// SIMATIC S7-200 project (STEP 7-Micro/WIN), CPU 224 REL 01.11

SYMBOL_TABLE USER1
Onn              I0.0
Off              I0.1
END_SYMBOL_TABLE

ORGANIZATION_BLOCK MAIN:OB1
TITLE=PROGRAM COMMENTS
BEGIN
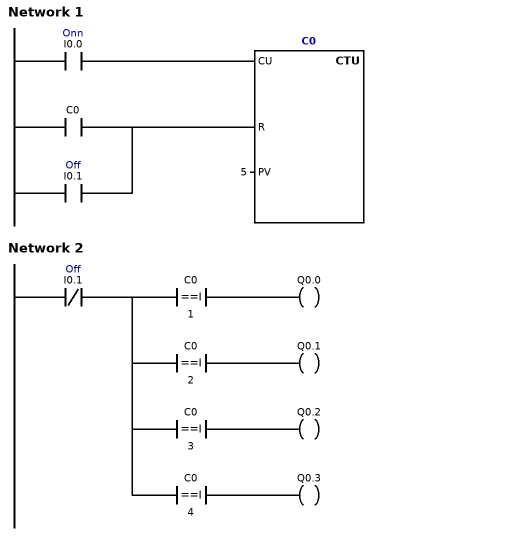
Network 1
LD     Onn:I0.0
LD     C0
O      Off:I0.1
CTU    C0, 5
Network 2
LDN    Off:I0.1
LPS
AW=    C0, 1
=      Q0.0
LRD
AW=    C0, 2
=      Q0.1
LRD
AW=    C0, 3
=      Q0.2
LPP
AW=    C0, 4
=      Q0.3
END_ORGANIZATION_BLOCK
